% RSLogix 500 project PV6.RSS, saved by version 8.30.00.16 %
PROJECT "PV6"    % processor: Bul.1763 MicroLogix 1100 Series B %

PROGRAM FILES
  LAD 2   30 rungs

DATA FILES
  O0 OUTPUT  5 elements
  I1 INPUT  7 elements
  S2 STATUS  66 elements
  B3 BINARY  2 elements
  T4 TIMER  3 elements
  C5 COUNTER  1 elements
  R6 CONTROL  1 elements
  N7 INTEGER  3 elements
  F8 FLOAT  1 elements

LADDER 2
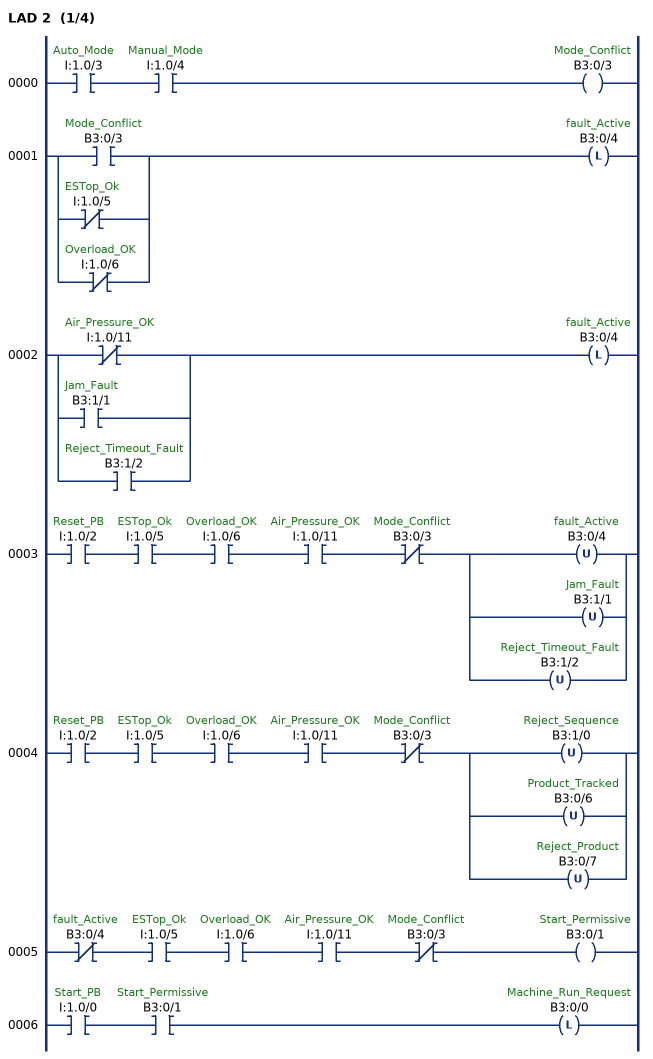
% Rung: 0 %
SOR XIC I:1.0/3 XIC I:1.0/4 OTE B3:0/3 EOR
%   I:1.0/3  "Auto_Mode" %
%   I:1.0/4  "Manual_Mode" %
%   B3:0/3  "Mode_Conflict" %
% Rung: 1 %
SOR BST XIC B3:0/3 NXB BST XIO I:1.0/5 NXB XIO I:1.0/6 BND BND OTL B3:0/4 EOR
%   B3:0/3  "Mode_Conflict" %
%   I:1.0/5  "ESTop_Ok" %
%   I:1.0/6  "Overload_OK" %
%   B3:0/4  "fault_Active" %
% Rung: 2 %
SOR BST XIO I:1.0/11 NXB BST XIC B3:1/1 NXB XIC B3:1/2 BND BND OTL B3:0/4 EOR
%   I:1.0/11  "Air_Pressure_OK" %
%   B3:1/1  "Jam_Fault" %
%   B3:1/2  "Reject_Timeout_Fault" %
%   B3:0/4  "fault_Active" %
% Rung: 3 %
SOR XIC I:1.0/2 XIC I:1.0/5 XIC I:1.0/6 XIC I:1.0/11 XIO B3:0/3 BST OTU B3:0/4 NXB BST OTU B3:1/1 NXB OTU B3:1/2 BND BND EOR
%   I:1.0/2  "Reset_PB" %
%   I:1.0/5  "ESTop_Ok" %
%   I:1.0/6  "Overload_OK" %
%   I:1.0/11  "Air_Pressure_OK" %
%   B3:0/3  "Mode_Conflict" %
%   B3:0/4  "fault_Active" %
%   B3:1/1  "Jam_Fault" %
%   B3:1/2  "Reject_Timeout_Fault" %
% Rung: 4 %
SOR XIC I:1.0/2 XIC I:1.0/5 XIC I:1.0/6 XIC I:1.0/11 XIO B3:0/3 BST OTU B3:1/0 NXB BST OTU B3:0/6 NXB OTU B3:0/7 BND BND EOR
%   I:1.0/2  "Reset_PB" %
%   I:1.0/5  "ESTop_Ok" %
%   I:1.0/6  "Overload_OK" %
%   I:1.0/11  "Air_Pressure_OK" %
%   B3:0/3  "Mode_Conflict" %
%   B3:1/0  "Reject_Sequence" %
%   B3:0/6  "Product_Tracked" %
%   B3:0/7  "Reject_Product" %
% Rung: 5 %
SOR XIO B3:0/4 XIC I:1.0/5 XIC I:1.0/6 XIC I:1.0/11 XIO B3:0/3 OTE B3:0/1 EOR
%   B3:0/4  "fault_Active" %
%   I:1.0/5  "ESTop_Ok" %
%   I:1.0/6  "Overload_OK" %
%   I:1.0/11  "Air_Pressure_OK" %
%   B3:0/3  "Mode_Conflict" %
%   B3:0/1  "Start_Permissive" %
% Rung: 6 %
SOR XIC I:1.0/0 XIC B3:0/1 OTL B3:0/0 EOR
%   I:1.0/0  "Start_PB" %
%   B3:0/1  "Start_Permissive" %
%   B3:0/0  "Machine_Run_Request" %

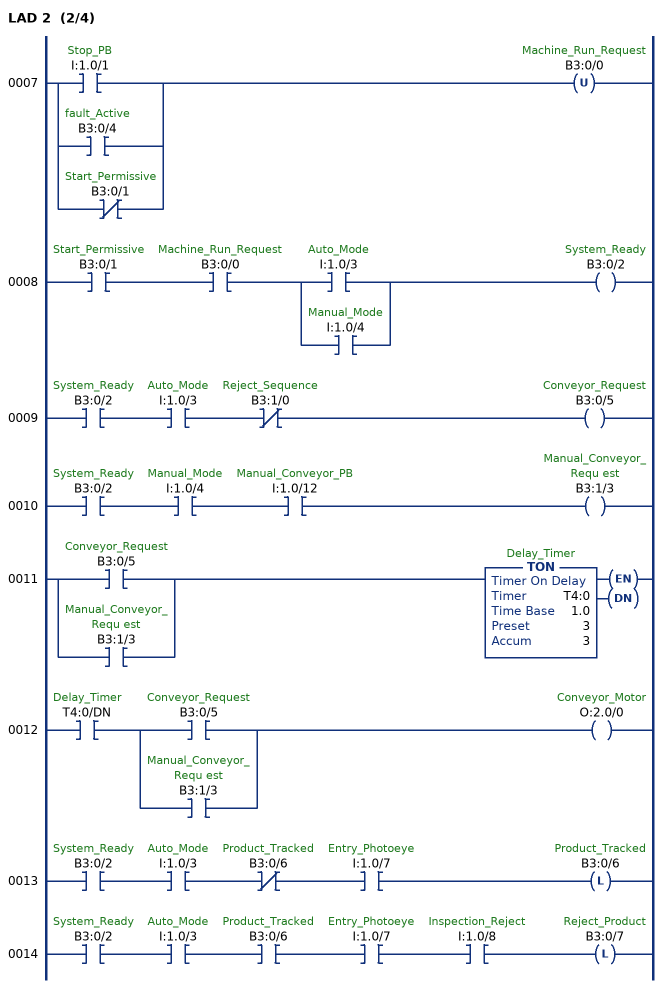
% Rung: 7 %
SOR BST XIC I:1.0/1 NXB BST XIC B3:0/4 NXB XIO B3:0/1 BND BND OTU B3:0/0 EOR
%   I:1.0/1  "Stop_PB" %
%   B3:0/4  "fault_Active" %
%   B3:0/1  "Start_Permissive" %
%   B3:0/0  "Machine_Run_Request" %
% Rung: 8 %
SOR XIC B3:0/1 XIC B3:0/0 BST XIC I:1.0/3 NXB XIC I:1.0/4 BND OTE B3:0/2 EOR
%   B3:0/1  "Start_Permissive" %
%   B3:0/0  "Machine_Run_Request" %
%   I:1.0/3  "Auto_Mode" %
%   I:1.0/4  "Manual_Mode" %
%   B3:0/2  "System_Ready" %
% Rung: 9 %
SOR XIC B3:0/2 XIC I:1.0/3 XIO B3:1/0 OTE B3:0/5 EOR
%   B3:0/2  "System_Ready" %
%   I:1.0/3  "Auto_Mode" %
%   B3:1/0  "Reject_Sequence" %
%   B3:0/5  "Conveyor_Request" %
% Rung: 10 %
SOR XIC B3:0/2 XIC I:1.0/4 XIC I:1.0/12 OTE B3:1/3 EOR
%   B3:0/2  "System_Ready" %
%   I:1.0/4  "Manual_Mode" %
%   I:1.0/12  "Manual_Conveyor_PB" %
%   B3:1/3  "Manual_Conveyor_Requ est" %
% Rung: 11 %
SOR BST XIC B3:0/5 NXB XIC B3:1/3 BND TON T4:0 1.0 3 3 EOR
%   B3:0/5  "Conveyor_Request" %
%   B3:1/3  "Manual_Conveyor_Requ est" %
%   T4:0  "Delay_Timer" %
% Rung: 12 %
SOR XIC T4:0/DN BST XIC B3:0/5 NXB XIC B3:1/3 BND OTE O:2.0/0 EOR
%   T4:0  "Delay_Timer" %
%   B3:0/5  "Conveyor_Request" %
%   B3:1/3  "Manual_Conveyor_Requ est" %
%   O:2.0/0  "Conveyor_Motor" %
% Rung: 13 %
SOR XIC B3:0/2 XIC I:1.0/3 XIO B3:0/6 XIC I:1.0/7 OTL B3:0/6 EOR
%   B3:0/2  "System_Ready" %
%   I:1.0/3  "Auto_Mode" %
%   B3:0/6  "Product_Tracked" %
%   I:1.0/7  "Entry_Photoeye" %
% Rung: 14 %
SOR XIC B3:0/2 XIC I:1.0/3 XIC B3:0/6 XIC I:1.0/7 XIC I:1.0/8 OTL B3:0/7 EOR
%   B3:0/2  "System_Ready" %
%   I:1.0/3  "Auto_Mode" %
%   B3:0/6  "Product_Tracked" %
%   I:1.0/7  "Entry_Photoeye" %
%   I:1.0/8  "Inspection_Reject" %
%   B3:0/7  "Reject_Product" %

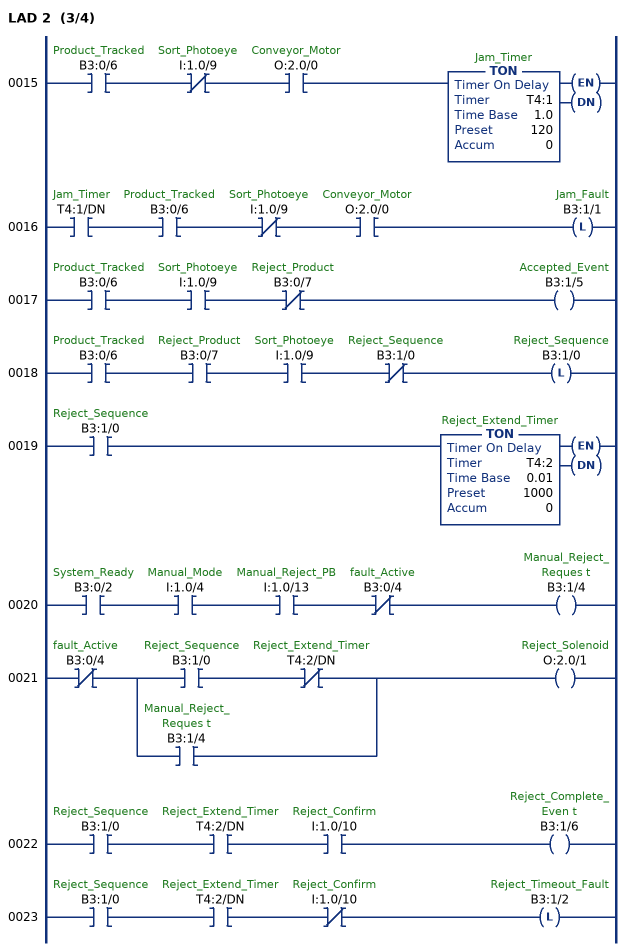
% Rung: 15 %
SOR XIC B3:0/6 XIO I:1.0/9 XIC O:2.0/0 TON T4:1 1.0 120 0 EOR
%   B3:0/6  "Product_Tracked" %
%   I:1.0/9  "Sort_Photoeye" %
%   O:2.0/0  "Conveyor_Motor" %
%   T4:1  "Jam_Timer" %
% Rung: 16 %
SOR XIC T4:1/DN XIC B3:0/6 XIO I:1.0/9 XIC O:2.0/0 OTL B3:1/1 EOR
%   T4:1  "Jam_Timer" %
%   B3:0/6  "Product_Tracked" %
%   I:1.0/9  "Sort_Photoeye" %
%   O:2.0/0  "Conveyor_Motor" %
%   B3:1/1  "Jam_Fault" %
% Rung: 17 %
SOR XIC B3:0/6 XIC I:1.0/9 XIO B3:0/7 OTE B3:1/5 EOR
%   B3:0/6  "Product_Tracked" %
%   I:1.0/9  "Sort_Photoeye" %
%   B3:0/7  "Reject_Product" %
%   B3:1/5  "Accepted_Event" %
% Rung: 18 %
SOR XIC B3:0/6 XIC B3:0/7 XIC I:1.0/9 XIO B3:1/0 OTL B3:1/0 EOR
%   B3:0/6  "Product_Tracked" %
%   B3:0/7  "Reject_Product" %
%   I:1.0/9  "Sort_Photoeye" %
%   B3:1/0  "Reject_Sequence" %
% Rung: 19 %
SOR XIC B3:1/0 TON T4:2 0.01 1000 0 EOR
%   B3:1/0  "Reject_Sequence" %
%   T4:2  "Reject_Extend_Timer" %
% Rung: 20 %
SOR XIC B3:0/2 XIC I:1.0/4 XIC I:1.0/13 XIO B3:0/4 OTE B3:1/4 EOR
%   B3:0/2  "System_Ready" %
%   I:1.0/4  "Manual_Mode" %
%   I:1.0/13  "Manual_Reject_PB" %
%   B3:0/4  "fault_Active" %
%   B3:1/4  "Manual_Reject_Reques t" %
% Rung: 21 %
SOR XIO B3:0/4 BST XIC B3:1/0 XIO T4:2/DN NXB XIC B3:1/4 BND OTE O:2.0/1 EOR
%   B3:0/4  "fault_Active" %
%   B3:1/0  "Reject_Sequence" %
%   T4:2  "Reject_Extend_Timer" %
%   B3:1/4  "Manual_Reject_Reques t" %
%   O:2.0/1  "Reject_Solenoid" %
% Rung: 22 %
SOR XIC B3:1/0 XIC T4:2/DN XIC I:1.0/10 OTE B3:1/6 EOR
%   B3:1/0  "Reject_Sequence" %
%   T4:2  "Reject_Extend_Timer" %
%   I:1.0/10  "Reject_Confirm" %
%   B3:1/6  "Reject_Complete_Even t" %
% Rung: 23 %
SOR XIC B3:1/0 XIC T4:2/DN XIO I:1.0/10 OTL B3:1/2 EOR
%   B3:1/0  "Reject_Sequence" %
%   T4:2  "Reject_Extend_Timer" %
%   I:1.0/10  "Reject_Confirm" %
%   B3:1/2  "Reject_Timeout_Fault" %

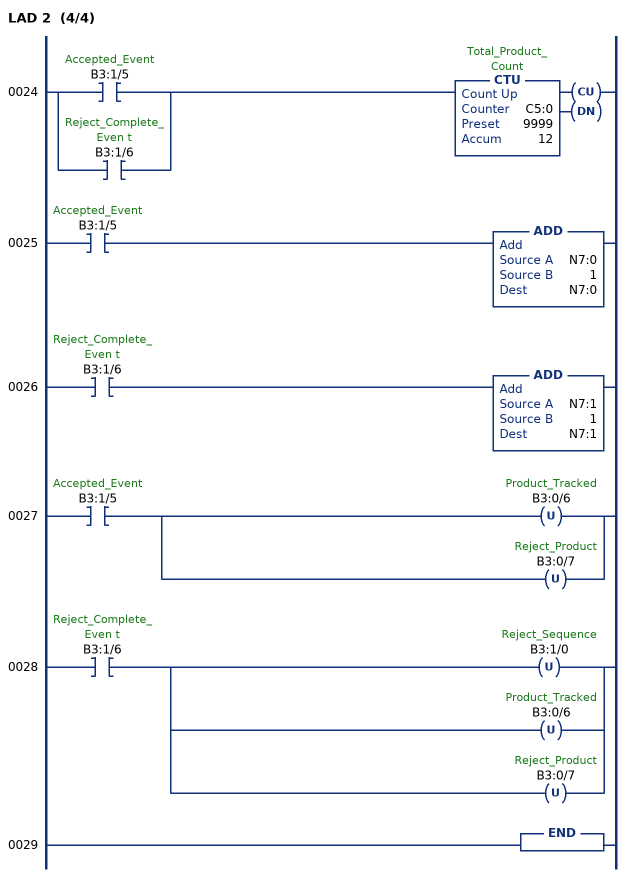
% Rung: 24 %
SOR BST XIC B3:1/5 NXB XIC B3:1/6 BND CTU C5:0 9999 12 EOR
%   B3:1/5  "Accepted_Event" %
%   B3:1/6  "Reject_Complete_Even t" %
%   C5:0  "Total_Product_Count" %
% Rung: 25 %
SOR XIC B3:1/5 ADD N7:0 1 N7:0 EOR
%   B3:1/5  "Accepted_Event" %
% Rung: 26 %
SOR XIC B3:1/6 ADD N7:1 1 N7:1 EOR
%   B3:1/6  "Reject_Complete_Even t" %
% Rung: 27 %
SOR XIC B3:1/5 BST OTU B3:0/6 NXB OTU B3:0/7 BND EOR
%   B3:1/5  "Accepted_Event" %
%   B3:0/6  "Product_Tracked" %
%   B3:0/7  "Reject_Product" %
% Rung: 28 %
SOR XIC B3:1/6 BST OTU B3:1/0 NXB BST OTU B3:0/6 NXB OTU B3:0/7 BND BND EOR
%   B3:1/6  "Reject_Complete_Even t" %
%   B3:1/0  "Reject_Sequence" %
%   B3:0/6  "Product_Tracked" %
%   B3:0/7  "Reject_Product" %
% Rung: 29 %
SOR END EOR

OTHER DOCUMENTED ADDRESSES
  C5:1  "Accepted_Count"
  I:3.0/0  "High_Level_Switch"
  O:2.0/2  "Cap_Solenoid"
  O:2.0/3  "Running_Lamp"
  O:2.0/4  "Fault_Lamp"
  O:2.0/5  "Alarm_Horn"
  T4:3  "Reject_Confirm_Timer"

DATA TABLE (non-zero values as saved)
DATA B3
% B3:0 % 0X0027 0X0000
DATA T4
% .PRE .ACC %
% T4:0 % 3 3
% T4:1 % 120 0
% T4:2 % 1000 0
DATA C5
% .PRE .ACC %
% C5:0 % 9999 12
DATA N7
% N7:0 % 1928 2 75
